TYPE ST_PISTON :
STRUCT
	ePISTON_TYPE: E_PISTON_TYPE;
	nNAME: STRING;
	openTime: REAL:=5;
	closeTime: REAL:=5;
	timeoutOpen:  TIME:=T#5S;
	timeoutClose: TIME:=T#5S;
	bOPEN_BY_DEFAULT: BOOL:= FALSE;
	
	
END_STRUCT
	
END_TYPE

(* stored: Version 1.1.0.1, ProductVersion 3.1.4024.12
   DUT ST_PISTON: Id {596ea6ff-1ac5-4a54-ab7a-469b15184d7d} *)
